// TwinCAT 3 PLC project PLC
// ProgramVersion: 3.1.4024.0
// libraries:
//   Tc2_Standard, * (Beckhoff Automation GmbH)
//   Tc2_System, * (Beckhoff Automation GmbH)
//   Tc3_Module, * (Beckhoff Automation GmbH)
//   VisuSymbols,3.5.10.0,System
// project tree:
//   DUTs/ PumpState.TcDUT, PumpStation.TcDUT, PumpType.TcDUT
//   / GlobalTextList.TcGTLO, PlcTask.TcTTO, Visualization Manager.TcVMO (not stored), Visualization.TcVIS
//   GVLs/ GVL.TcGVL
//   POUs/ AlternatePump.TcPOU, FindAndStartPump.TcPOU, FindAndStopPump.TcPOU, LevelControl.TcPOU, MAIN.TcPOU, NoOfRunningPumps.TcPOU, StartPump.TcPOU, StopPump.TcPOU, UpdateCounters.TcPOU
// real-time tasks:
//   TASK PlcTask: cycle T#10ms, priority 20, ADS port 350

CONFIGURATION PLC
    RESOURCE PLC ON TwinCAT3
        TASK PlcTask(INTERVAL := T#10ms, PRIORITY := 20);
        PROGRAM MAIN WITH PlcTask : MAIN;
    END_RESOURCE
END_CONFIGURATION

// ---- DUTs/PumpState.TcDUT
{attribute 'qualified_only'}
{attribute 'strict'}
TYPE PumpState :
	(STOP, RUN, ALARM, SERVICE):= STOP;
END_TYPE

// ---- DUTs/PumpStation.TcDUT
TYPE PumpStation :
STRUCT
	PumpsArray				:	ARRAY[1..GVL.MAX_PUMPS] OF PumpType;
	NoPumpsRun				:	INT;	// number of running pumps
	Level					:	WORD;	// water level in the tank
END_STRUCT
END_TYPE

// ---- DUTs/PumpType.TcDUT
TYPE PumpType :
STRUCT
	RunState				:	PumpState := PumpState.STOP;
	RunTotalMinutes			:	DWORD:=0;
	RunLastStartSec			:	WORD:=0;
	RunSeconds				:	WORD:=0;	// count up to 60
	RunTimerSeconds			:	TON;		// count up RunSeconds
END_STRUCT
END_TYPE

// ---- GVLs/GVL.TcGVL
{attribute 'qualified_only'}
VAR_GLOBAL CONSTANT
	MAX_PUMPS: BYTE:=6;
END_VAR

// ---- POUs/MAIN.TcPOU
PROGRAM MAIN
VAR
	PumpTank			:	PumpStation;			// one pump station ceontains all pumps
END_VAR

// update counters
UpdateCounters(Pumps:=PumpTank.PumpsArray);

// pump alternating time is 3600 seconds = 1 hour.
// can be changed to a lower time  when testing
AlternatePump(AlternationTimeSec:=10, PumpTank:=PumpTank);

// update nomber of running pumps
PumpTank.NoPumpsRun := NoOfRunningPumps(Pumps:=PumpTank.PumpsArray);

// find the required pumps to run depending on the level in the tank
LevelControl(751, 1000, 6, PumpTank); 
LevelControl(601, 750, 5, PumpTank);
LevelControl(451, 600, 4, PumpTank);
LevelControl(301, 450, 3, PumpTank);
LevelControl(151, 300, 2, PumpTank);
LevelControl(100, 150, 1, PumpTank);
LevelControl(0, 99, 0, PumpTank);

END_PROGRAM

// ---- POUs/UpdateCounters.TcPOU
FUNCTION UpdateCounters : BOOL
VAR_IN_OUT
	Pumps		:	ARRAY[1..GVL.MAX_PUMPS] of PumpType;
END_VAR
VAR
	Idx			:	INT;		// loop counter
END_VAR

FOR Idx := 1 TO GVL.MAX_PUMPS DO
	Pumps[Idx].RunTimerSeconds(IN:=NOT Pumps[Idx].RunTimerSeconds.Q, PT:=T#1S);
	
	// only update when pump in RUN state
	IF Pumps[Idx].RunState = PumpState.RUN THEN
		
		// check if second timer ended
		IF Pumps[Idx].RunTimerSeconds.Q THEN
			Pumps[Idx].RunSeconds := Pumps[Idx].RunSeconds + 1;
			Pumps[Idx].RunLastStartSec := Pumps[Idx].RunLastStartSec + 1;

			// update minutes
			IF Pumps[Idx].RunSeconds >= 60 THEN
				Pumps[Idx].RunTotalMinutes := Pumps[Idx].RunTotalMinutes + 1;
				Pumps[Idx].RunSeconds:=0; 
			END_IF
 
		END_IF
	END_IF
END_FOR

END_FUNCTION

// ---- POUs/AlternatePump.TcPOU
FUNCTION AlternatePump : BOOL
VAR_INPUT
	AlternationTimeSec	:	DWORD;			// time a pump has to run before alternating
END_VAR
VAR_IN_OUT
	PumpTank			:	PumpStation;	// address pointer to the STRUCT outside the function
END_VAR
VAR
	Idx					:	INT;			// loop index
END_VAR

(*
FC for alternating between pumps.   
AlternationTimeSec -  Time until pump alternation
*)

// only alternate between pumps if at least one, but not all pumps are running
IF PumpTank.NoPumpsRun > 0 THEN
	IF PumpTank.NoPumpsRun < GVL.MAX_PUMPS THEN
		// check all pumps
		FOR Idx:=1 TO GVL.MAX_PUMPS DO
			IF AlternationTimeSec<PumpTank.PumpsArray[Idx].RunLastStartSec AND
			   PumpTank.PumpsArray[Idx].RunState=PumpState.RUN THEN
				  
			  // first stop the pump that is running for the longest time
			  StopPump(Pump:=PumpTank.PumpsArray[Idx]);
			  
			  // then start another pump
			  FindAndStartPump(Pumps:=PumpTank.PumpsArray);
			  
			EXIT;	// only alternate to one pump. Another pump will be checked in next scan
			END_IF
			
		END_FOR
	END_IF
END_IF

END_FUNCTION

// ---- POUs/StopPump.TcPOU
FUNCTION StopPump : BOOL
VAR_IN_OUT
	Pump		:	PumpType;
END_VAR
VAR
END_VAR

// pump will stop after 30 sec delay to avoid unnecessary start/stop

IF Pump.RunLastStartSec > 5 THEN
	Pump.RunState := PumpState.STOP;
	Pump.RunLastStartSec := 0;
END_IF

END_FUNCTION

// ---- POUs/FindAndStartPump.TcPOU
FUNCTION FindAndStartPump : BOOL
VAR_IN_OUT
	Pumps		:	ARRAY[1..GVL.MAX_PUMPS] OF PumpType;
END_VAR
VAR
	Idx			:	INT;
	RunTime		:	DWORD;
	PumpIndex	:	INT;
END_VAR

RunTime := 9999999;			// set initial high tiem to find a low run time
PumpIndex := 1;

// find a pump in stop state with the lowest run time
FOR Idx:=1 TO GVL.MAX_PUMPS DO
	IF RunTime > Pumps[Idx].RunTotalMinutes AND Pumps[Idx].RunState=PumpState.STOP THEN
		RunTime:=Pumps[Idx].RunTotalMinutes;
		PumpIndex:=Idx;
	END_IF
END_FOR

// start pump
StartPump(Pump:=Pumps[PumpIndex]);

END_FUNCTION

// ---- POUs/StartPump.TcPOU
FUNCTION StartPump : BOOL
VAR_IN_OUT
	Pump	:	PumpType;
END_VAR
VAR
END_VAR

// start pump
Pump.RunState := Pumpstate.RUN;

END_FUNCTION

// ---- POUs/NoOfRunningPumps.TcPOU
FUNCTION NoOfRunningPumps : INT
VAR_IN_OUT
	Pumps		:	ARRAY[1..GVL.MAX_PUMPS] OF PumpType;
END_VAR
VAR
	Idx			:	INT;
	No			:	INT:=0;	// counter of running pumps
END_VAR

(* 
Count number of running pumps
*)

FOR Idx:=1 TO GVL.MAX_PUMPS DO
	IF Pumps[Idx].RunState = PumpState.RUN THEN
		No:=No+1;
	END_IF
END_FOR

NoOfRunningPumps := No;

END_FUNCTION

// ---- POUs/LevelControl.TcPOU
FUNCTION LevelControl : BOOL
VAR_INPUT
	LevelLow			:	WORD;		// liquid level in tank must be above this level
	LevelHigh			:	WORD;		// liquid level in tank must be belove this level
	NoPumpsReq			:	INT;		// number of pumps required to run in the liquid level range
END_VAR
VAR_IN_OUT
	PumpTank			:	PumpStation;	// address pointer to the STRUCT outside the function
END_VAR
VAR
	PumpControl			:	INT:=0;		
END_VAR

(*
This FC starts or stops a pump depending on the level in the tank
*)

// check level. Does a pump need to be started due to a high liquid level?
IF PumpTank.Level>=LevelLow AND PumpTank.Level<=LevelHigh THEN
	IF NoPumpsReq>PumpTank.NoPumpsRun THEN
		// negative if one more pump needed
		PumpControl:=NoPumpsReq-PumpTank.NoPumpsRun;
	END_IF
END_IF

// check level. Does a pump need to be stopped due to a low liquid level?
IF PumpTank.Level>=LevelLow AND PumpTank.Level<=LevelHigh THEN
	IF NoPumpsReq<PumpTank.NoPumpsRun THEN
		// positivve if a pump has to be stopped
		PumpControl := NoPumpsReq-PumpTank.NoPumpsRun; 
	END_IF
END_IF

// stop a pump if needed
IF PumpControl<0 THEN
	FindAndStopPump(Pumps:=PumpTank.PumpsArray);
END_IF

// start a pump if needed
IF PumpControl>0 THEN
	FindAndStartPump(Pumps:=PumpTank.PumpsArray);
END_IF

END_FUNCTION

// ---- POUs/FindAndStopPump.TcPOU
FUNCTION FindAndStopPump : BOOL
VAR_IN_OUT
	Pumps			:	ARRAY[1..GVL.MAX_PUMPS] OF PumpType;
END_VAR
VAR
	Idx				:	INT;
	RunTime			:	DWORD;
	PumpIndex		:	INT;
END_VAR

// set an initial lwo time to find the highest run time
RunTime := 0;
PumpIndex := 0;


// find the pump in run state with the longest accumulated run time
FOR Idx := 1 TO GVL.MAX_PUMPS DO
	IF RunTime < Pumps[Idx].RunTotalMinutes AND Pumps[Idx].RunState = PumpState.RUN THEN
		RunTime := Pumps[Idx].RunTotalMinutes;
		PumpIndex := Idx;
	END_IF
END_FOR

// stop the pump
IF PumpIndex > 0 AND PumpIndex <= GVL.MAX_PUMPS THEN
	StopPump(Pump:=Pumps[PumpIndex]);
END_IF

END_FUNCTION

// ---- GlobalTextList.TcGTLO
TEXTLIST GlobalTextList
  410 = '1'
  963 = '2'
  13 = '3'
  34 = '4'
  740 = '5'
  75 = '6'
  969 = 'Pump 1'
  781 = 'Tank level'
END_TEXTLIST

// ---- Visualization.TcVIS
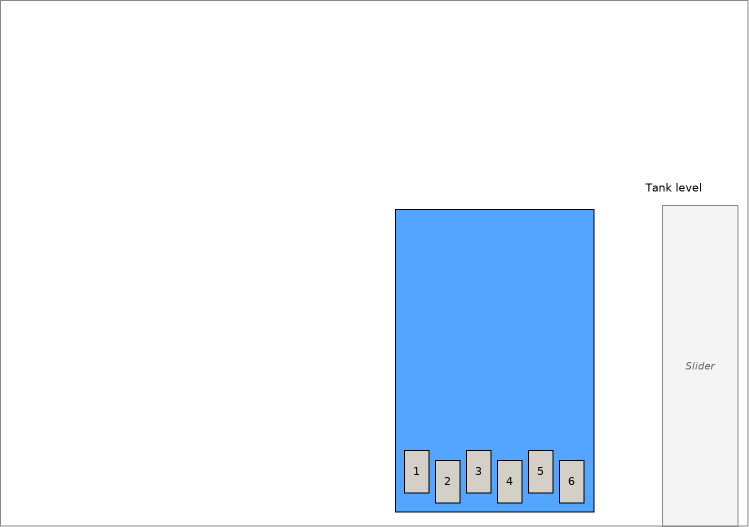
VISUALIZATION Visualization  // 749x527
    Rectangle (395,209 199x303)
    RoundedRectangle (404,450 25x43), "1", colour toggle: MAIN.PumpTank.PumpsArray[1].RunState=PumpState.RUN
    RoundedRectangle (435,460 25x43), "2", colour toggle: MAIN.PumpTank.PumpsArray[2].RunState=PumpState.RUN
    RoundedRectangle (466,450 25x43), "3", colour toggle: MAIN.PumpTank.PumpsArray[3].RunState=PumpState.RUN
    RoundedRectangle (497,460 25x43), "4", colour toggle: MAIN.PumpTank.PumpsArray[4].RunState=PumpState.RUN
    RoundedRectangle (559,460 25x43), "6", colour toggle: MAIN.PumpTank.PumpsArray[6].RunState=PumpState.RUN
    RoundedRectangle (528,450 25x43), "5", colour toggle: MAIN.PumpTank.PumpsArray[5].RunState=PumpState.RUN
    Slider (662,205 76x322), variable: MAIN.PumpTank.Level, scale 0..1000
    Label (599,173 150x30), "Tank level"
END_VISUALIZATION
